(* PLC project Generated.project, CODESYS CODESYS V3.5 SP19 Patch 1 *)
(* stored: creationDateTime 2026-08-27T21:37:02.540638, modificationDateTime 2026-08-27T21:37:02.540638 *)

(* ======================================================================= 🪣 ST_fbCycle_BucketCmdDemand — Demande de commande benne ─────────────────────────────────────────────────────────────── 🎯 Rôle : Structure de consigne de mouvement benne (Ouverture, Fermeture, Kobold) 📄 Doc métier : DOC/AF/AF_Partie-10_Fonction_Winch_v2.1.md ======================================================================= *)
TYPE ST_fbCycle_BucketCmdDemand : STRUCT
  Open : BOOL;  (* Demande ouverture benne *)
  Close : BOOL;  (* Demande fermeture benne *)
  KoboldContactorCmd : BOOL;  (* Commande contacteur puissance Kobold (recherche fond) *)
END_STRUCT;
END_TYPE
